FUNCTION_BLOCK Read_FLOAT (* Template for a Simple Function Block Type *)
  (* Standard: 61499-1 *)
  (* Version 1.0, 2024-07-26, david *)
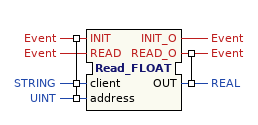
  EVENT_INPUT
    INIT WITH client, address; (* Initialization event *)
    READ; (* Read event *)
  END_EVENT
  EVENT_OUTPUT
    INIT_O; (* Init event out *)
    READ_O WITH OUT; (* Read event out *)
  END_EVENT
  VAR_INPUT
    client : STRING; (* client object *)
    address : UINT; (* register address *)
  END_VAR
  VAR_OUTPUT
    OUT : REAL; (* Output *)
  END_VAR
END_FUNCTION_BLOCK
(* other elements stored in the file *)
(* With Var=client *)
(* With Var=address *)
